// TwinCAT 3 PLC project PLC
// ProgramVersion: 3.1.4024.0
// libraries:
//   Tc2_Standard, * (Beckhoff Automation GmbH)
//   Tc2_System, * (Beckhoff Automation GmbH)
//   Tc3_Module, * (Beckhoff Automation GmbH)
// project tree:
//   / GlobalTextList.TcGTLO, PlcTask.TcTTO, Visu1.TcVIS, Visualization Manager.TcVMO (not stored)
//   POUs/ Fifo.TcPOU, MAIN.TcPOU
// real-time tasks:
//   TASK PlcTask: cycle T#10ms, priority 20, ADS port 350

CONFIGURATION PLC
    RESOURCE PLC ON TwinCAT3
        TASK PlcTask(INTERVAL := T#10ms, PRIORITY := 20);
        PROGRAM MAIN WITH PlcTask : MAIN;
    END_RESOURCE
END_CONFIGURATION

// ---- POUs/MAIN.TcPOU
PROGRAM MAIN
VAR
	ItemCode			:	STRING(10);
	ItemNo				:	INT;
	
	tonIn				:	TON;
	ton01				:	TON;
	ton02				:	TON;
	ton03				:	TON;
	ton04				:	TON;
	
	tpIn				:	TP;
	tpM02In				:	TP;
	tpM03In				:	TP;
	tpM02Out			:	TP;
	tpM03Out			:	TP;
	tpM04Out			:	TP;
	tpEolOut			:	TP;
	Eol					:	BOOL;
	rtrigEol			:	R_TRIG;
	
	Fifo01				:	Fifo;
	Fifo02				:	Fifo;
	Fifo03				:	Fifo;
	Fifo04				:	Fifo;
	FifoEol				:	Fifo;

END_VAR

// simulation for item inlet
tonIn(IN:=NOT tonIn.Q, PT:=T#1600MS);

// simulation for machine processing M1,M2,M3,M4
ton01(IN:=NOT ton01.Q, PT:=T#3S);
ton02(IN:=NOT ton02.Q, PT:=T#8S);
ton03(IN:=NOT ton03.Q, PT:=T#6S);
ton04(IN:=NOT ton04.Q, PT:=T#7S);

// enf of line test ok
rtrigEol(CLK:=Eol);


Fifo01(QueueLength:=10);	// FIFO for M1
Fifo02(QueueLength:=10);	// FIFO for M2
Fifo03(QueueLength:=10);	// FIFO for M3
Fifo04(QueueLength:=10);	// FIFO for M4
FifoEol(QueueLength:=10);	// FIFO for End of Line station

// timers for visualisation
tpIn(PT:=T#500MS);
tpIn.IN:=FALSE;

tpM02In(PT:=T#500MS);
tpM02In.IN:=FALSE;

tpM03In(PT:=T#500MS);
tpM03In.IN:=FALSE;

tpM02Out(PT:=T#500MS);
tpM02Out.IN:=FALSE;

tpM03Out(PT:=T#500MS);
tpM03Out.IN:=FALSE;

tpM04Out(PT:=T#500MS);
tpM04Out.IN:=FALSE;

tpEolOut(PT:=T#500MS);
tpEolOut.IN:=FALSE;
	

// item inlet into M1
IF tonIn.Q AND NOT Fifo01.IsFull THEN
	tpIn.IN := tonIn.Q;
	// move item into M1 if buffer not full
	ItemNo:=ItemNo+1;
	ItemCode:=CONCAT('ITEM',INT_TO_STRING(ItemNo));
	Fifo01.InsertToQueue(DataIn:=ItemCode);	
END_IF


// M1 out
IF ton01.Q AND NOT Fifo01.IsEmpty THEN
	IF Fifo02.NoOfDataPoints<Fifo03.NoOfDataPoints AND NOT Fifo02.IsFull THEN
		// move item to M2
		Fifo02.InsertToQueue(DataIn:=Fifo01.RemoveFromQueue());
		tpM02In.IN:=ton01.Q;
	ELSIF Fifo03.NoOfDataPoints<Fifo02.NoOfDataPoints AND NOT Fifo03.IsFull THEN
		// move item to M3
		Fifo03.InsertToQueue(DataIn:=Fifo01.RemoveFromQueue());
		tpM03In.IN:=ton01.Q;
	ELSIF Fifo02.NoOfDataPoints=Fifo03.NoOfDataPoints AND NOT Fifo03.IsFull THEN
		// move item to M3 (M3 has faster processing time) 
		Fifo03.InsertToQueue(DataIn:=Fifo01.RemoveFromQueue());
		tpM03In.IN:=ton01.Q;
	END_IF
END_IF

// M2 out
IF ton02.Q AND NOT Fifo02.IsEmpty THEN
	IF NOT Fifo04.IsFull THEN
		Fifo04.InsertToQueue(DataIn:=Fifo02.RemoveFromQueue());
		tpM02Out.IN:=ton02.Q;
	END_IF
END_IF


// M3 out
IF ton03.Q AND NOT Fifo03.IsEmpty THEN
	IF NOT Fifo04.IsFull THEN
		Fifo04.InsertToQueue(DataIn:=Fifo03.RemoveFromQueue());
		tpM03Out.IN:=ton03.Q;
	END_IF
END_IF


// M4 out
IF ton04.Q AND NOT Fifo04.IsEmpty THEN 
	IF NOT FifoEol.IsFull THEN
		FifoEol.InsertToQueue(DataIn:=Fifo04.RemoveFromQueue());
		tpM04Out.IN:=ton04.Q;
	END_IF
END_IF

// M5 out
IF rtrigEol.Q AND NOT FifoEol.IsEmpty THEN
	FifoEol.RemoveFromQueue();
	tpEolOut.IN:=rtrigEol.Q;
END_IF

END_PROGRAM

// ---- POUs/Fifo.TcPOU
FUNCTION_BLOCK Fifo
VAR_INPUT
	QueueLength			:	INT;
END_VAR

VAR_OUTPUT
	ErrorMsg			:	STRING(50);	// error message
	QueueFull			:	Bool;
	QueueEmpty			:	BOOL;
END_VAR

VAR CONSTANT
	QueueMin			: 	INT:=0;
	QueueMax			:	INT:=29;
END_VAR

VAR
	ptrHead				:	INT ;		// pointer to first element (head)
	ptrTail				:	INT ; 		// pointer to last element (tail) 
	Idx					:	INT;
	InitBit				:	BOOL:=TRUE;
	QueueSize			:	INT;		// size of circular queue
	QueueSizeOk			:	BOOL;		
	Queue				:	ARRAY[QueueMin..QueueMax] OF STRING(10);
END_VAR

(*
This FB acts as FIFO i.e. circular queue.
Size of the queue must be customized with constants QueueMin and QueueMax. 
*)
IF InitBit THEN

	InitBit := FALSE;
	
	IF QueueMax > QueueMin AND QueueLength>1 THEN
		ErrorMsg:='';
		ptrHead := -1;
		ptrTail := -1;
		QueueSize := TO_INT(SIZEOF(Queue) / SIZEOF(REAL));
		QueueSizeOk := TRUE;
	ELSE
		QueueSizeOk:=FALSE;
		ErrorMsg:='Queue Length must be > 1';
	END_IF
END_IF

METHOD ClearQueue : BOOL
VAR_INPUT
END_VAR
// reinit the queue

IF QueueSizeOk THEN
	ptrHead := -1;
	ptrTail := -1;
	
	FOR Idx := QueueMin TO QueueMax DO
		Queue[Idx] := '';
	END_FOR

	ErrorMsg := '';
	QueueEmpty := FALSE;
	QueueFull := FALSE;
END_IF
END_METHOD

METHOD InsertToQueue : BOOL
VAR_INPUT
	DataIn		:	STRING(10);			// data to insert into circular queue
END_VAR
// Insert new data into queue

IF QueueSizeOk THEN 
	IF IsFull THEN
		// queue is full. can't insert new data
		ErrorMsg := 'Queue is full. Can not insert new data';
		QueueFull := TRUE;
	ELSIF IsEmpty THEN
		ErrorMsg := '';
		QueueFull := FALSE;
		ptrHead := 0;
		ptrTail := 0;
		Queue[ptrTail] := DataIn;
	ELSE 
		ErrorMsg := '';
		QueueFull := FALSE;
		IF (ptrTail+1) MOD QueueLength <= QueueLength THEN
			ptrTail := (ptrTail + 1) MOD QueueLength;
			Queue[ptrTail] := DataIn;	
		END_IF
	
	END_IF
END_IF
END_METHOD

PROPERTY IsEmpty : BOOL
GET
IsEmpty := ptrHead = -1 AND ptrTail = -1;
END_GET
END_PROPERTY

PROPERTY IsFull : BOOL
GET
IsFull := ptrHead = (ptrTail + 1) MOD QueueLength;
END_GET
END_PROPERTY

PROPERTY NoOfDataPoints : INT
GET
// number of data points in queue
IF ptrTail>ptrHead THEN
	NoOfDataPoints:=ABS(ptrTail - ptrHead)+1;
ELSIF ptrTail<ptrHead THEN
	NoOfDataPoints:=(ptrTail+1) + (QueueLength-ptrHead);
ELSE
	// ptrTail=ptrHead
	NoOfDataPoints:=0;
END_IF
END_GET
END_PROPERTY

METHOD RemoveFromQueue : STRING(10);
VAR_INPUT
END_VAR
// remove one data from the queue

IF QueueSizeOk THEN
	IF IsEmpty THEN							// zero element in queue
		ErrorMsg := 'Queue is empty';
		QueueEmpty := TRUE;
	ELSIF ptrHead=ptrTail THEN				// only one element in queue
		ErrorMsg := '';
		QueueEmpty := FALSE;
		RemoveFromQueue := Queue[ptrHead];
		Queue[ptrHead]:='';
		ptrHead := -1;
		ptrTail := -1;
	ELSE									// more then one element in queue
		ErrorMsg := '';
		QueueEmpty := FALSE;
		IF (ptrHead + 1) MOD QueueLength <= QueueLength THEN
			RemoveFromQueue := Queue[ptrHead];
			Queue[ptrHead]:='';
			ptrHead := (ptrHead + 1) MOD QueueLength;
		END_IF
	END_IF
END_IF
END_METHOD

END_FUNCTION_BLOCK

// ---- GlobalTextList.TcGTLO
TEXTLIST GlobalTextList
  140 = 'End of Line Test'
  411 = 'End of Line Test\nEOL'
  912 = 'EOL Test OK'
  309 = 'Item Inlet'
  489 = 'Item Outlet'
  192 = 'Machine 1\nM1'
  718 = 'Machine 2\nM2'
  527 = 'Machine 3\nM3'
  998 = 'Machine 4\nM4'
  263 = 'Queue'
END_TEXTLIST

// ---- Visu1.TcVIS
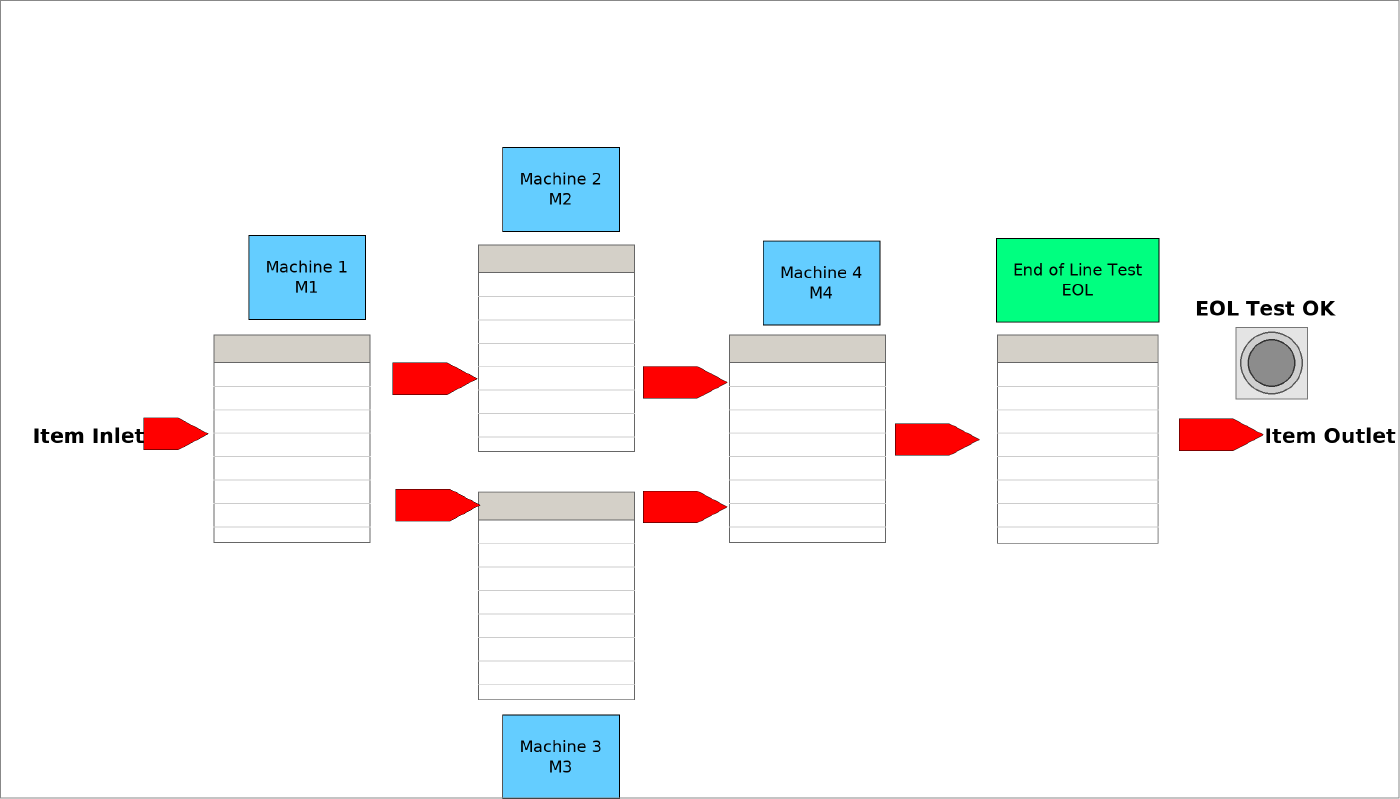
VISUALIZATION Visu1  // 1494x853
    Table (228,357 167x222), data array: MAIN.Fifo01.Queue
        p3854506369: MAIN.Fifo01.Queue[INDEX]
        p2232123230: FIFO_TEST.Fifo01.Queue[INDEX]
    Table (510,261 167x221), data array: MAIN.Fifo02.Queue
        p3854506369: MAIN.Fifo02.Queue[INDEX]
        p2232123230: FIFO_TEST.Fifo02.Queue[INDEX]
    Table (510,525 167x222), data array: MAIN.Fifo03.Queue
        p3854506369: MAIN.Fifo03.Queue[INDEX]
        p2232123230: FIFO_TEST.Fifo03.Queue[INDEX]
    Table (778,357 167x222), data array: MAIN.Fifo04.Queue
        p3854506369: MAIN.Fifo04.Queue[INDEX]
        p2232123230: FIFO_TEST.Fifo04.Queue[INDEX]
    Table (1064,357 172x223), data array: MAIN.FifoEol.Queue
        p3854506369: MAIN.FifoEol.Queue[INDEX]
        p2232123230: FIFO_TEST.Fifo05.Queue[INDEX]
    PushSwitch (1315,349 84x77), variable: MAIN.Eol, behaviour: TAP, style: Switch-PushSwitch-Gray
    Polygon (153,446) (153,480) (190,480) (222,463) (190,446), invisible if: NOT MAIN.tpIn.Q
    Polygon (419,387) (419,421) (477,421) (509,404) (477,387), invisible if: NOT MAIN.tpM02In.Q
    Polygon (422,522) (422,556) (480,556) (512,539) (480,522), invisible if: NOT MAIN.tpM03In.Q
    Polygon (686,391) (686,425) (744,425) (776,408) (744,391), invisible if: NOT MAIN.tpM02Out.Q
    Polygon (686,524) (686,558) (744,558) (776,541) (744,524), invisible if: NOT MAIN.tpM03Out.Q
    Polygon (955,452) (955,486) (1013,486) (1045,469) (1013,452), invisible if: NOT MAIN.tpM04Out.Q
    Polygon (1258,447) (1258,481) (1316,481) (1348,464) (1316,447), invisible if: NOT MAIN.tpEolOut.Q
    RoundedRectangle (265,251 125x90), "Machine 1 M1"
    RoundedRectangle (536,157 125x90), "Machine 2 M2"
    RoundedRectangle (536,763 125x90), "Machine 3 M3"
    RoundedRectangle (814,257 125x90), "Machine 4 M4"
    RoundedRectangle (1063,254 174x90), "End of Line Test EOL"
    Label (1264,308 172x43), "EOL Test OK"
    Label (20,444 149x43), "Item Inlet"
    Label (1345,444 149x43), "Item Outlet"
END_VISUALIZATION
